KUKA KRL program: ProfileHeight.src, ProfileHeight.dat

--- ProfileHeight.src ---
&ACCESS RV1
&REL 12
DEFFCT REAL ProfileHeight(eProfile:IN)
   DECL E_ProfileType eProfile
   DECL REAL rProfileZ

   SWITCH eProfile
      CASE #Frame75
         rProfileZ = rFrame75
      CASE #Frame90
         rProfileZ = rFrame90
      CASE #Leaf75
         rProfileZ = rLeaf75
      CASE #Leaf90
         rProfileZ = rLeaf90
      CASE #Threshold75
         rProfileZ = rThreshold75
      CASE #Threshold90
         rProfileZ = rThreshold90
      DEFAULT
         HALT
   ENDSWITCH

   RETURN rProfileZ

ENDFCT

--- ProfileHeight.dat ---
&ACCESS RV1
&REL 12
DEFDAT ProfileHeight

   DECL CONST REAL rFrame75 = 70.0
   DECL CONST REAL rLeaf75 = 67.4
   DECL CONST REAL rThreshold75 = 18.5

   DECL CONST REAL rFrame90 = 70.4
   DECL CONST REAL rLeaf90 = 51.0
   DECL CONST REAL rThreshold90 = 18.0

ENDDAT
